// TIA Portal V17 export
// export: Created 2023-12-22T15:05:24.9190485Z, ExportSetting WithDefaults, DisplayName Totally Integrated Automation Portal, DisplayVersion V17, DisplayName TIA Portal Openness, DisplayVersion V17, DisplayName TIA Portal Version Control Interface, DisplayVersion V17, DisplayName STEP 7 Professional, DisplayVersion V17, DisplayName STEP 7 Safety, DisplayVersion V17, DisplayName WinCC Advanced, DisplayVersion V17
FUNCTION "Line_Settings" : Void   // FC2, LAD
{ S7_Optimized_Access := 'TRUE' }
VERSION : 0.1
// stored: AutoNumber true, IsIECCheckEnabled false, SetENOAutomatically false, UDAEnableTagReadback false
   VAR_INPUT
      All_lines : Int;   // Кол-во линий
   END_VAR
   VAR_IN_OUT
      Line_REQ : Int;   // Запрос линии
      Line_Now : Int;   // Линия сейчас
      Ready : Bool;   // Готовность
   END_VAR
   VAR_TEMP   // added for the SCL form of the ladder/FBD networks
      _w1 : Bool;
      _w2 : Bool;
      _w3 : Bool;
      _w4 : Bool;
      _w5 : Bool;
      _w6 : Bool;
      _w7 : Bool;
      _w8 : Bool;
      _w9 : Bool;
   END_VAR
BEGIN

REGION Network 1: Проверка корректности выбранной линии
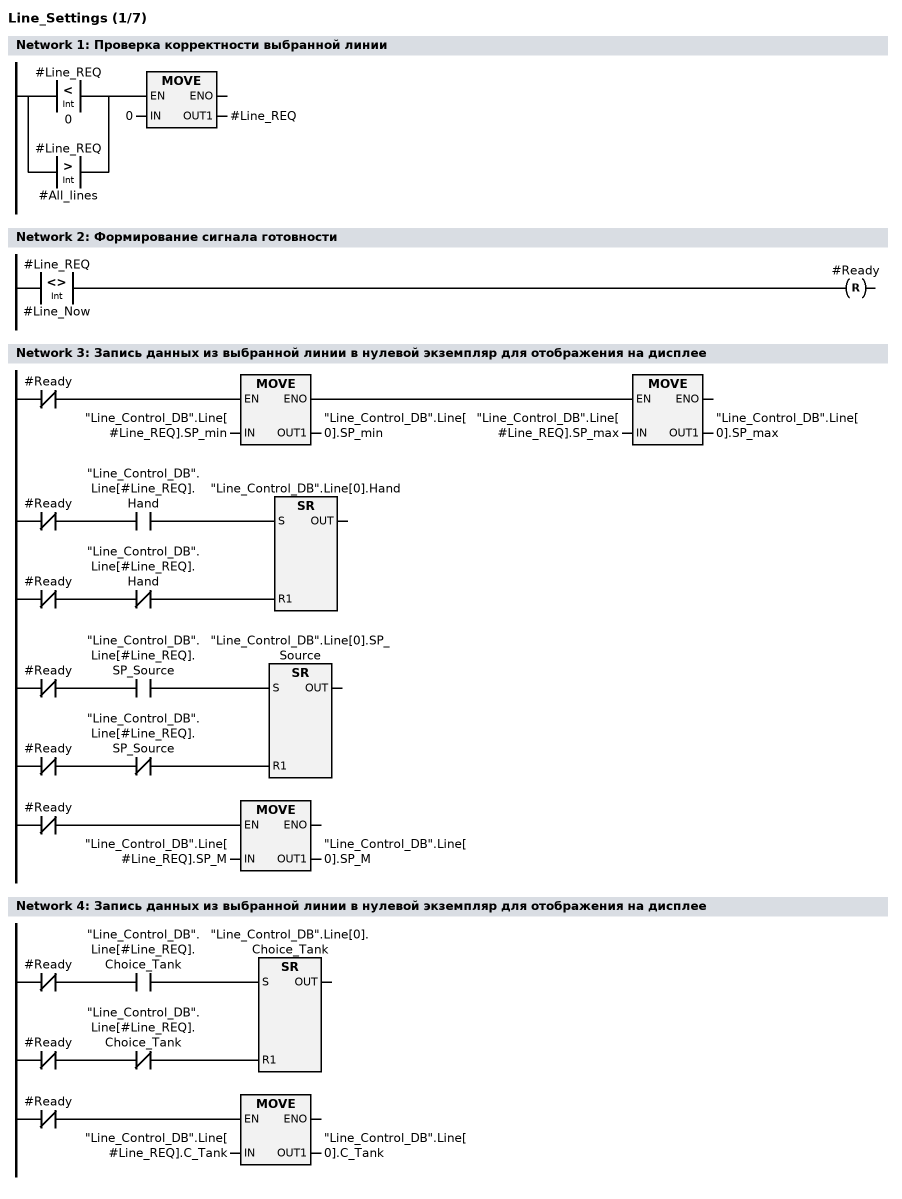
   RUNG wire#powerrail
      { S7_Templates := "SrcType := Int" } LT_Contact(in1 := #Line_REQ, in2 := 0)
      wire#w1
      Move(in := 0, out1 => #Line_REQ)
   END_RUNG
   RUNG wire#powerrail
      { S7_Templates := "SrcType := Int" } GT_Contact(in1 := #Line_REQ, in2 := #All_lines)
   END_RUNG wire#w1
   // the same network as SCL:
   IF (#Line_REQ < 0) OR (#Line_REQ > #All_lines) THEN #Line_REQ := 0; END_IF;
END_REGION

REGION Network 2: Формирование сигнала готовности
   RUNG wire#powerrail
      { S7_Templates := "SrcType := Int" } NE_Contact(in1 := #Line_REQ, in2 := #Line_Now)
      R_Coil( #Ready )
   END_RUNG
   // the same network as SCL:
   IF #Line_REQ <> #Line_Now THEN #Ready := FALSE; END_IF;
END_REGION

REGION Network 3: Запись данных из выбранной линии в нулевой экземпляр для отображения на дисплее
   RUNG wire#powerrail
      I_Contact( #Ready )
      Move(in := "Line_Control_DB".Line[#Line_REQ].SP_min, out1 => "Line_Control_DB".Line[0].SP_min)
      Move(in := "Line_Control_DB".Line[#Line_REQ].SP_max, out1 => "Line_Control_DB".Line[0].SP_max)
   END_RUNG
   RUNG wire#powerrail
      I_Contact( #Ready )
      Contact( "Line_Control_DB".Line[#Line_REQ].Hand )
      S_SR(operand := "Line_Control_DB".Line[0].Hand, r1 := wire#w1)
   END_RUNG
   RUNG wire#powerrail
      I_Contact( #Ready )
      I_Contact( "Line_Control_DB".Line[#Line_REQ].Hand )
   END_RUNG wire#w1
   RUNG wire#powerrail
      I_Contact( #Ready )
      Contact( "Line_Control_DB".Line[#Line_REQ].SP_Source )
      S_SR(operand := "Line_Control_DB".Line[0].SP_Source, r1 := wire#w2)
   END_RUNG
   RUNG wire#powerrail
      I_Contact( #Ready )
      I_Contact( "Line_Control_DB".Line[#Line_REQ].SP_Source )
   END_RUNG wire#w2
   RUNG wire#powerrail
      I_Contact( #Ready )
      Move(in := "Line_Control_DB".Line[#Line_REQ].SP_M, out1 => "Line_Control_DB".Line[0].SP_M)
   END_RUNG
   // the same network as SCL:
   IF NOT #Ready THEN
       "Line_Control_DB".Line[0].SP_min := "Line_Control_DB".Line[#Line_REQ].SP_min;
       "Line_Control_DB".Line[0].SP_max := "Line_Control_DB".Line[#Line_REQ].SP_max;
   END_IF;
   #_w1 := NOT #Ready AND NOT "Line_Control_DB".Line[#Line_REQ].Hand;
   IF NOT #Ready AND "Line_Control_DB".Line[#Line_REQ].Hand THEN
       "Line_Control_DB".Line[0].Hand := TRUE;   // SR flip-flop
   END_IF;
   IF #_w1 THEN "Line_Control_DB".Line[0].Hand := FALSE; END_IF;
   #_w2 := NOT #Ready AND NOT "Line_Control_DB".Line[#Line_REQ].SP_Source;
   IF NOT #Ready AND "Line_Control_DB".Line[#Line_REQ].SP_Source THEN
       "Line_Control_DB".Line[0].SP_Source := TRUE;   // SR flip-flop
   END_IF;
   IF #_w2 THEN "Line_Control_DB".Line[0].SP_Source := FALSE; END_IF;
   IF NOT #Ready THEN "Line_Control_DB".Line[0].SP_M := "Line_Control_DB".Line[#Line_REQ].SP_M; END_IF;
END_REGION

REGION Network 4: Запись данных из выбранной линии в нулевой экземпляр для отображения на дисплее
   RUNG wire#powerrail
      I_Contact( #Ready )
      Contact( "Line_Control_DB".Line[#Line_REQ].Choice_Tank )
      S_SR(operand := "Line_Control_DB".Line[0].Choice_Tank, r1 := wire#w1)
   END_RUNG
   RUNG wire#powerrail
      I_Contact( #Ready )
      I_Contact( "Line_Control_DB".Line[#Line_REQ].Choice_Tank )
   END_RUNG wire#w1
   RUNG wire#powerrail
      I_Contact( #Ready )
      Move(in := "Line_Control_DB".Line[#Line_REQ].C_Tank, out1 => "Line_Control_DB".Line[0].C_Tank)
   END_RUNG
   // the same network as SCL:
   #_w1 := NOT #Ready AND NOT "Line_Control_DB".Line[#Line_REQ].Choice_Tank;
   IF NOT #Ready AND "Line_Control_DB".Line[#Line_REQ].Choice_Tank THEN
       "Line_Control_DB".Line[0].Choice_Tank := TRUE;   // SR flip-flop
   END_IF;
   IF #_w1 THEN "Line_Control_DB".Line[0].Choice_Tank := FALSE; END_IF;
   IF NOT #Ready THEN "Line_Control_DB".Line[0].C_Tank := "Line_Control_DB".Line[#Line_REQ].C_Tank; END_IF;
END_REGION

REGION Network 5: Запись данных из выбранной линии в нулевой экземпляр для отображения на дисплее
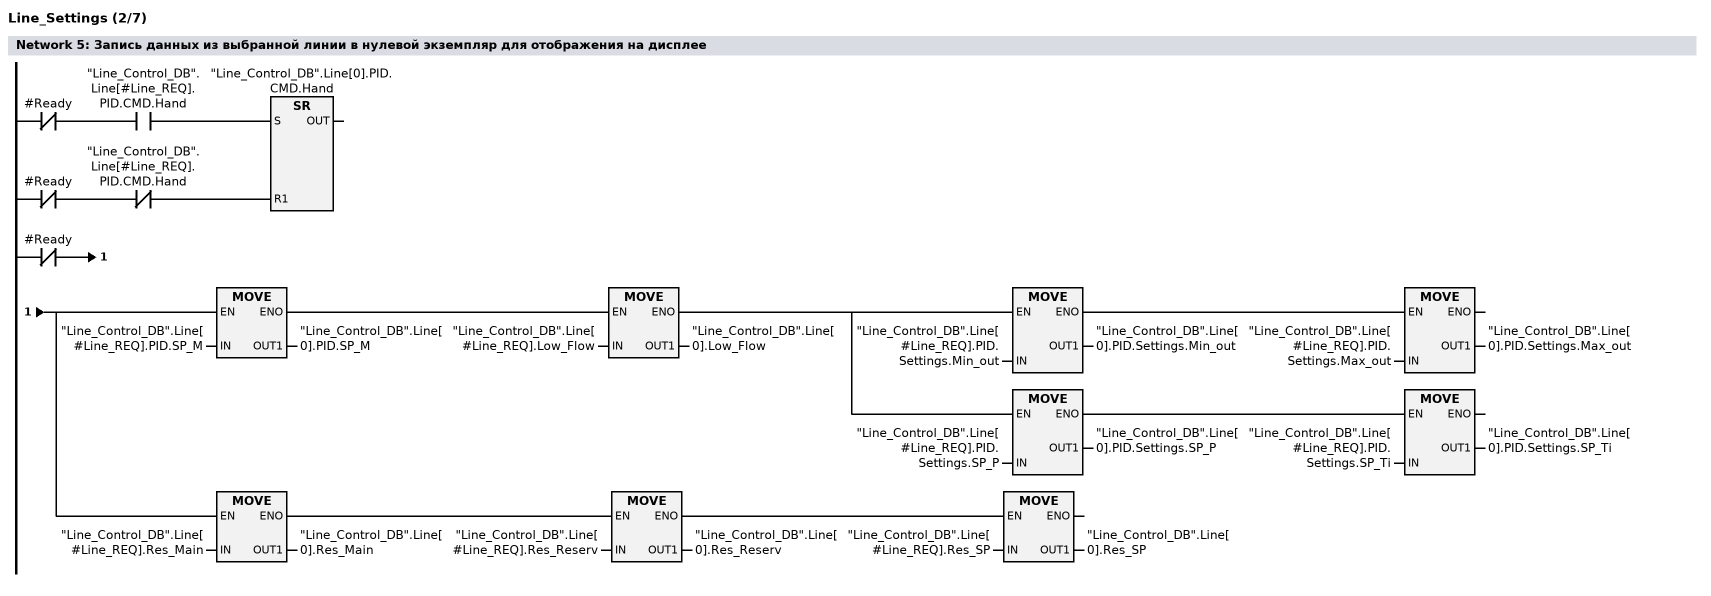
   RUNG wire#powerrail
      I_Contact( #Ready )
      Contact( "Line_Control_DB".Line[#Line_REQ].PID.CMD.Hand )
      S_SR(operand := "Line_Control_DB".Line[0].PID.CMD.Hand, r1 := wire#w1)
   END_RUNG
   RUNG wire#powerrail
      I_Contact( #Ready )
      I_Contact( "Line_Control_DB".Line[#Line_REQ].PID.CMD.Hand )
   END_RUNG wire#w1
   RUNG wire#powerrail
      I_Contact( #Ready )
      wire#w2
      Move(in := "Line_Control_DB".Line[#Line_REQ].PID.SP_M, out1 => "Line_Control_DB".Line[0].PID.SP_M)
      Move(in := "Line_Control_DB".Line[#Line_REQ].Low_Flow, out1 => "Line_Control_DB".Line[0].Low_Flow)
      wire#w3
      Move(in := "Line_Control_DB".Line[#Line_REQ].PID.Settings.Min_out, out1 => "Line_Control_DB".Line[0].PID.Settings.Min_out)
      Move(in := "Line_Control_DB".Line[#Line_REQ].PID.Settings.Max_out, out1 => "Line_Control_DB".Line[0].PID.Settings.Max_out)
   END_RUNG
   RUNG wire#w3
      Move(in := "Line_Control_DB".Line[#Line_REQ].PID.Settings.SP_P, out1 => "Line_Control_DB".Line[0].PID.Settings.SP_P)
      Move(in := "Line_Control_DB".Line[#Line_REQ].PID.Settings.SP_Ti, out1 => "Line_Control_DB".Line[0].PID.Settings.SP_Ti)
   END_RUNG
   RUNG wire#w2
      Move(in := "Line_Control_DB".Line[#Line_REQ].Res_Main, out1 => "Line_Control_DB".Line[0].Res_Main)
      Move(in := "Line_Control_DB".Line[#Line_REQ].Res_Reserv, out1 => "Line_Control_DB".Line[0].Res_Reserv)
      Move(in := "Line_Control_DB".Line[#Line_REQ].Res_SP, out1 => "Line_Control_DB".Line[0].Res_SP)
   END_RUNG
   // the same network as SCL:
   #_w1 := NOT #Ready AND NOT "Line_Control_DB".Line[#Line_REQ].PID.CMD.Hand;
   IF NOT #Ready AND "Line_Control_DB".Line[#Line_REQ].PID.CMD.Hand THEN
       "Line_Control_DB".Line[0].PID.CMD.Hand := TRUE;   // SR flip-flop
   END_IF;
   IF #_w1 THEN "Line_Control_DB".Line[0].PID.CMD.Hand := FALSE; END_IF;
   IF NOT #Ready THEN
       "Line_Control_DB".Line[0].PID.SP_M := "Line_Control_DB".Line[#Line_REQ].PID.SP_M;
       "Line_Control_DB".Line[0].Low_Flow := "Line_Control_DB".Line[#Line_REQ].Low_Flow;
       "Line_Control_DB".Line[0].PID.Settings.Min_out := "Line_Control_DB".Line[#Line_REQ].PID.Settings.Min_out;
       "Line_Control_DB".Line[0].PID.Settings.Max_out := "Line_Control_DB".Line[#Line_REQ].PID.Settings.Max_out;
       "Line_Control_DB".Line[0].PID.Settings.SP_P := "Line_Control_DB".Line[#Line_REQ].PID.Settings.SP_P;
       "Line_Control_DB".Line[0].PID.Settings.SP_Ti := "Line_Control_DB".Line[#Line_REQ].PID.Settings.SP_Ti;
       "Line_Control_DB".Line[0].Res_Main := "Line_Control_DB".Line[#Line_REQ].Res_Main;
       "Line_Control_DB".Line[0].Res_Reserv := "Line_Control_DB".Line[#Line_REQ].Res_Reserv;
       "Line_Control_DB".Line[0].Res_SP := "Line_Control_DB".Line[#Line_REQ].Res_SP;
   END_IF;
END_REGION

REGION Network 6: Запись данных из выбранной линии в нулевой экземпляр для отображения на дисплее
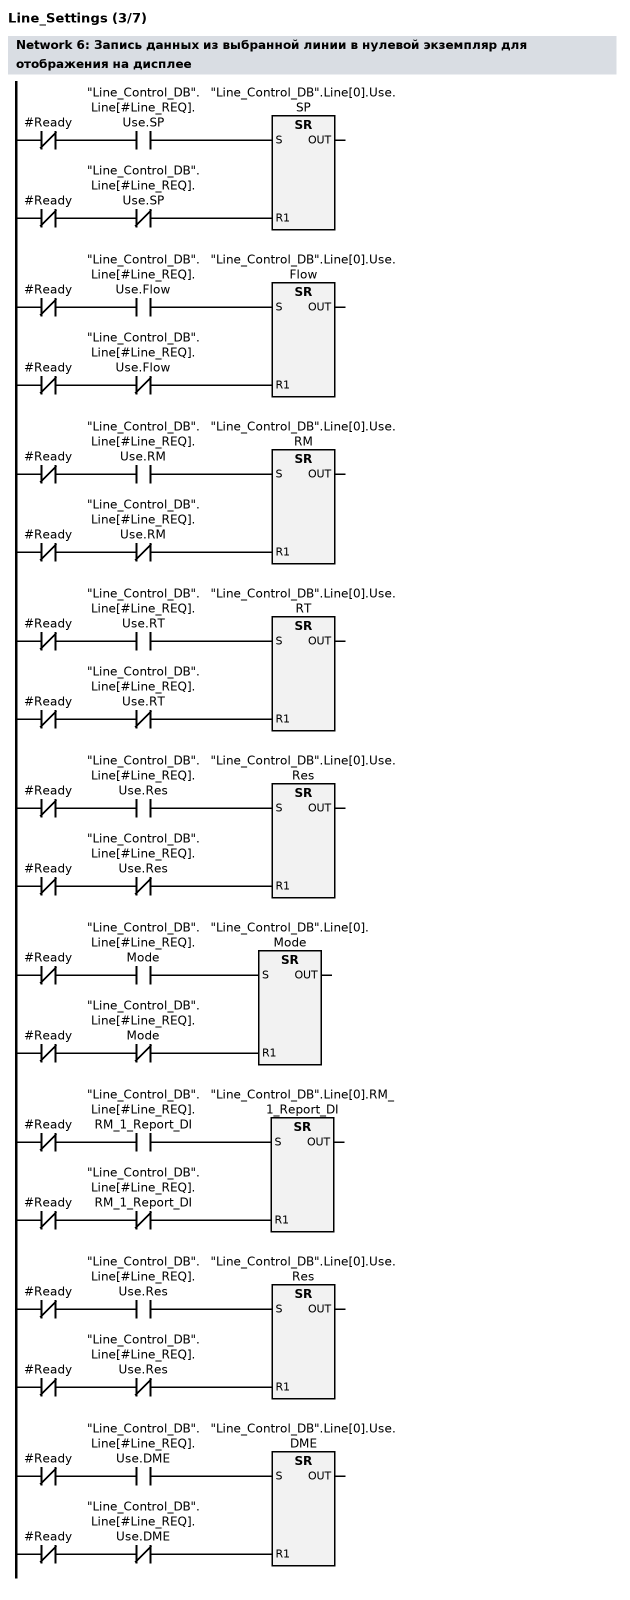
   RUNG wire#powerrail
      I_Contact( #Ready )
      Contact( "Line_Control_DB".Line[#Line_REQ].Use.SP )
      S_SR(operand := "Line_Control_DB".Line[0].Use.SP, r1 := wire#w1)
   END_RUNG
   RUNG wire#powerrail
      I_Contact( #Ready )
      I_Contact( "Line_Control_DB".Line[#Line_REQ].Use.SP )
   END_RUNG wire#w1
   RUNG wire#powerrail
      I_Contact( #Ready )
      Contact( "Line_Control_DB".Line[#Line_REQ].Use.Flow )
      S_SR(operand := "Line_Control_DB".Line[0].Use.Flow, r1 := wire#w2)
   END_RUNG
   RUNG wire#powerrail
      I_Contact( #Ready )
      I_Contact( "Line_Control_DB".Line[#Line_REQ].Use.Flow )
   END_RUNG wire#w2
   RUNG wire#powerrail
      I_Contact( #Ready )
      Contact( "Line_Control_DB".Line[#Line_REQ].Use.RM )
      S_SR(operand := "Line_Control_DB".Line[0].Use.RM, r1 := wire#w3)
   END_RUNG
   RUNG wire#powerrail
      I_Contact( #Ready )
      I_Contact( "Line_Control_DB".Line[#Line_REQ].Use.RM )
   END_RUNG wire#w3
   RUNG wire#powerrail
      I_Contact( #Ready )
      Contact( "Line_Control_DB".Line[#Line_REQ].Use.RT )
      S_SR(operand := "Line_Control_DB".Line[0].Use.RT, r1 := wire#w4)
   END_RUNG
   RUNG wire#powerrail
      I_Contact( #Ready )
      I_Contact( "Line_Control_DB".Line[#Line_REQ].Use.RT )
   END_RUNG wire#w4
   RUNG wire#powerrail
      I_Contact( #Ready )
      Contact( "Line_Control_DB".Line[#Line_REQ].Use.Res )
      S_SR(operand := "Line_Control_DB".Line[0].Use.Res, r1 := wire#w5)
   END_RUNG
   RUNG wire#powerrail
      I_Contact( #Ready )
      I_Contact( "Line_Control_DB".Line[#Line_REQ].Use.Res )
   END_RUNG wire#w5
   RUNG wire#powerrail
      I_Contact( #Ready )
      Contact( "Line_Control_DB".Line[#Line_REQ].Mode )
      S_SR(operand := "Line_Control_DB".Line[0].Mode, r1 := wire#w6)
   END_RUNG
   RUNG wire#powerrail
      I_Contact( #Ready )
      I_Contact( "Line_Control_DB".Line[#Line_REQ].Mode )
   END_RUNG wire#w6
   RUNG wire#powerrail
      I_Contact( #Ready )
      Contact( "Line_Control_DB".Line[#Line_REQ].RM_1_Report_DI )
      S_SR(operand := "Line_Control_DB".Line[0].RM_1_Report_DI, r1 := wire#w7)
   END_RUNG
   RUNG wire#powerrail
      I_Contact( #Ready )
      I_Contact( "Line_Control_DB".Line[#Line_REQ].RM_1_Report_DI )
   END_RUNG wire#w7
   RUNG wire#powerrail
      I_Contact( #Ready )
      Contact( "Line_Control_DB".Line[#Line_REQ].Use.Res )
      S_SR(operand := "Line_Control_DB".Line[0].Use.Res, r1 := wire#w8)
   END_RUNG
   RUNG wire#powerrail
      I_Contact( #Ready )
      I_Contact( "Line_Control_DB".Line[#Line_REQ].Use.Res )
   END_RUNG wire#w8
   RUNG wire#powerrail
      I_Contact( #Ready )
      Contact( "Line_Control_DB".Line[#Line_REQ].Use.DME )
      S_SR(operand := "Line_Control_DB".Line[0].Use.DME, r1 := wire#w9)
   END_RUNG
   RUNG wire#powerrail
      I_Contact( #Ready )
      I_Contact( "Line_Control_DB".Line[#Line_REQ].Use.DME )
   END_RUNG wire#w9
   // the same network as SCL:
   #_w1 := NOT #Ready AND NOT "Line_Control_DB".Line[#Line_REQ].Use.SP;
   IF NOT #Ready AND "Line_Control_DB".Line[#Line_REQ].Use.SP THEN
       "Line_Control_DB".Line[0].Use.SP := TRUE;   // SR flip-flop
   END_IF;
   IF #_w1 THEN "Line_Control_DB".Line[0].Use.SP := FALSE; END_IF;
   #_w2 := NOT #Ready AND NOT "Line_Control_DB".Line[#Line_REQ].Use.Flow;
   IF NOT #Ready AND "Line_Control_DB".Line[#Line_REQ].Use.Flow THEN
       "Line_Control_DB".Line[0].Use.Flow := TRUE;   // SR flip-flop
   END_IF;
   IF #_w2 THEN "Line_Control_DB".Line[0].Use.Flow := FALSE; END_IF;
   #_w3 := NOT #Ready AND NOT "Line_Control_DB".Line[#Line_REQ].Use.RM;
   IF NOT #Ready AND "Line_Control_DB".Line[#Line_REQ].Use.RM THEN
       "Line_Control_DB".Line[0].Use.RM := TRUE;   // SR flip-flop
   END_IF;
   IF #_w3 THEN "Line_Control_DB".Line[0].Use.RM := FALSE; END_IF;
   #_w4 := NOT #Ready AND NOT "Line_Control_DB".Line[#Line_REQ].Use.RT;
   IF NOT #Ready AND "Line_Control_DB".Line[#Line_REQ].Use.RT THEN
       "Line_Control_DB".Line[0].Use.RT := TRUE;   // SR flip-flop
   END_IF;
   IF #_w4 THEN "Line_Control_DB".Line[0].Use.RT := FALSE; END_IF;
   #_w5 := NOT #Ready AND NOT "Line_Control_DB".Line[#Line_REQ].Use.Res;
   IF NOT #Ready AND "Line_Control_DB".Line[#Line_REQ].Use.Res THEN
       "Line_Control_DB".Line[0].Use.Res := TRUE;   // SR flip-flop
   END_IF;
   IF #_w5 THEN "Line_Control_DB".Line[0].Use.Res := FALSE; END_IF;
   #_w6 := NOT #Ready AND NOT "Line_Control_DB".Line[#Line_REQ].Mode;
   IF NOT #Ready AND "Line_Control_DB".Line[#Line_REQ].Mode THEN
       "Line_Control_DB".Line[0].Mode := TRUE;   // SR flip-flop
   END_IF;
   IF #_w6 THEN "Line_Control_DB".Line[0].Mode := FALSE; END_IF;
   #_w7 := NOT #Ready AND NOT "Line_Control_DB".Line[#Line_REQ].RM_1_Report_DI;
   IF NOT #Ready AND "Line_Control_DB".Line[#Line_REQ].RM_1_Report_DI THEN
       "Line_Control_DB".Line[0].RM_1_Report_DI := TRUE;   // SR flip-flop
   END_IF;
   IF #_w7 THEN "Line_Control_DB".Line[0].RM_1_Report_DI := FALSE; END_IF;
   #_w8 := NOT #Ready AND NOT "Line_Control_DB".Line[#Line_REQ].Use.Res;
   IF NOT #Ready AND "Line_Control_DB".Line[#Line_REQ].Use.Res THEN
       "Line_Control_DB".Line[0].Use.Res := TRUE;   // SR flip-flop
   END_IF;
   IF #_w8 THEN "Line_Control_DB".Line[0].Use.Res := FALSE; END_IF;
   #_w9 := NOT #Ready AND NOT "Line_Control_DB".Line[#Line_REQ].Use.DME;
   IF NOT #Ready AND "Line_Control_DB".Line[#Line_REQ].Use.DME THEN
       "Line_Control_DB".Line[0].Use.DME := TRUE;   // SR flip-flop
   END_IF;
   IF #_w9 THEN "Line_Control_DB".Line[0].Use.DME := FALSE; END_IF;
END_REGION

REGION Network 7: Запись данных из выбранной линии в нулевой экземпляр для отображения на дисплее
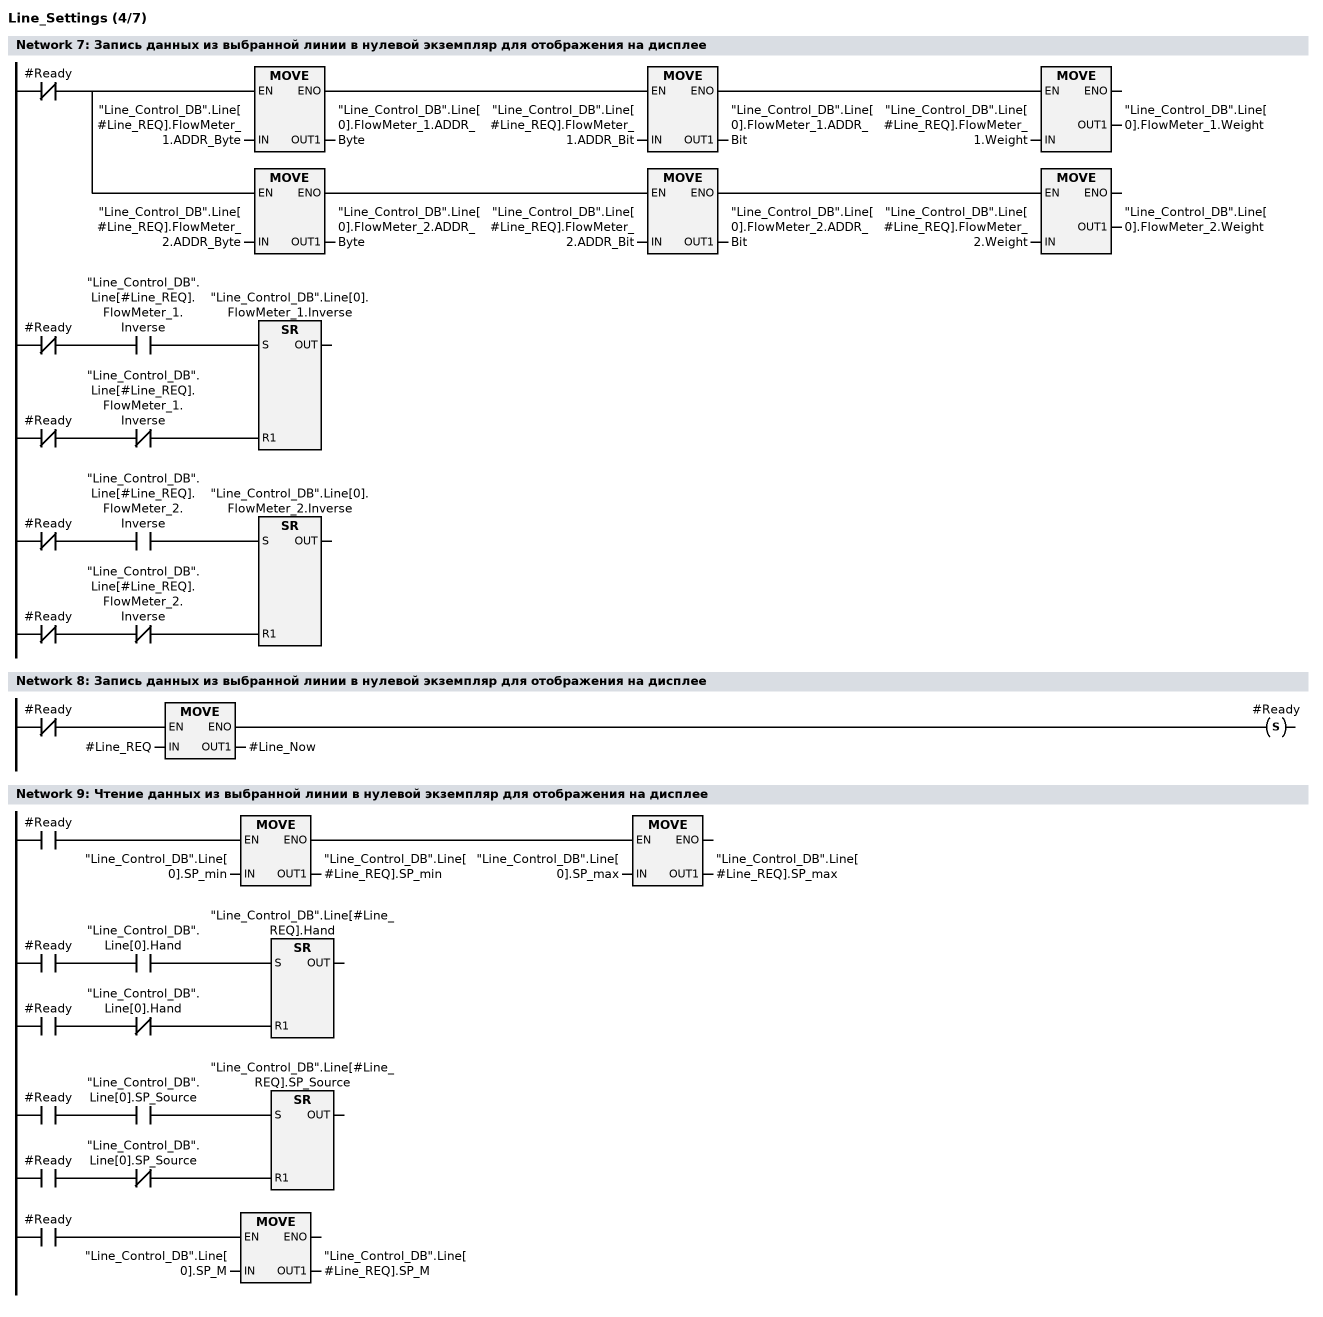
   RUNG wire#powerrail
      I_Contact( #Ready )
      wire#w1
      Move(in := "Line_Control_DB".Line[#Line_REQ].FlowMeter_1.ADDR_Byte, out1 => "Line_Control_DB".Line[0].FlowMeter_1.ADDR_Byte)
      Move(in := "Line_Control_DB".Line[#Line_REQ].FlowMeter_1.ADDR_Bit, out1 => "Line_Control_DB".Line[0].FlowMeter_1.ADDR_Bit)
      Move(in := "Line_Control_DB".Line[#Line_REQ].FlowMeter_1.Weight, out1 => "Line_Control_DB".Line[0].FlowMeter_1.Weight)
   END_RUNG
   RUNG wire#w1
      Move(in := "Line_Control_DB".Line[#Line_REQ].FlowMeter_2.ADDR_Byte, out1 => "Line_Control_DB".Line[0].FlowMeter_2.ADDR_Byte)
      Move(in := "Line_Control_DB".Line[#Line_REQ].FlowMeter_2.ADDR_Bit, out1 => "Line_Control_DB".Line[0].FlowMeter_2.ADDR_Bit)
      Move(in := "Line_Control_DB".Line[#Line_REQ].FlowMeter_2.Weight, out1 => "Line_Control_DB".Line[0].FlowMeter_2.Weight)
   END_RUNG
   RUNG wire#powerrail
      I_Contact( #Ready )
      Contact( "Line_Control_DB".Line[#Line_REQ].FlowMeter_1.Inverse )
      S_SR(operand := "Line_Control_DB".Line[0].FlowMeter_1.Inverse, r1 := wire#w2)
   END_RUNG
   RUNG wire#powerrail
      I_Contact( #Ready )
      I_Contact( "Line_Control_DB".Line[#Line_REQ].FlowMeter_1.Inverse )
   END_RUNG wire#w2
   RUNG wire#powerrail
      I_Contact( #Ready )
      Contact( "Line_Control_DB".Line[#Line_REQ].FlowMeter_2.Inverse )
      S_SR(operand := "Line_Control_DB".Line[0].FlowMeter_2.Inverse, r1 := wire#w3)
   END_RUNG
   RUNG wire#powerrail
      I_Contact( #Ready )
      I_Contact( "Line_Control_DB".Line[#Line_REQ].FlowMeter_2.Inverse )
   END_RUNG wire#w3
   // the same network as SCL:
   IF NOT #Ready THEN
       "Line_Control_DB".Line[0].FlowMeter_1.ADDR_Byte := "Line_Control_DB".Line[#Line_REQ].FlowMeter_1.ADDR_Byte;
       "Line_Control_DB".Line[0].FlowMeter_1.ADDR_Bit := "Line_Control_DB".Line[#Line_REQ].FlowMeter_1.ADDR_Bit;
       "Line_Control_DB".Line[0].FlowMeter_1.Weight := "Line_Control_DB".Line[#Line_REQ].FlowMeter_1.Weight;
       "Line_Control_DB".Line[0].FlowMeter_2.ADDR_Byte := "Line_Control_DB".Line[#Line_REQ].FlowMeter_2.ADDR_Byte;
       "Line_Control_DB".Line[0].FlowMeter_2.ADDR_Bit := "Line_Control_DB".Line[#Line_REQ].FlowMeter_2.ADDR_Bit;
       "Line_Control_DB".Line[0].FlowMeter_2.Weight := "Line_Control_DB".Line[#Line_REQ].FlowMeter_2.Weight;
   END_IF;
   #_w1 := NOT #Ready AND NOT "Line_Control_DB".Line[#Line_REQ].FlowMeter_1.Inverse;
   IF NOT #Ready AND "Line_Control_DB".Line[#Line_REQ].FlowMeter_1.Inverse THEN
       "Line_Control_DB".Line[0].FlowMeter_1.Inverse := TRUE;   // SR flip-flop
   END_IF;
   IF #_w1 THEN "Line_Control_DB".Line[0].FlowMeter_1.Inverse := FALSE; END_IF;
   #_w2 := NOT #Ready AND NOT "Line_Control_DB".Line[#Line_REQ].FlowMeter_2.Inverse;
   IF NOT #Ready AND "Line_Control_DB".Line[#Line_REQ].FlowMeter_2.Inverse THEN
       "Line_Control_DB".Line[0].FlowMeter_2.Inverse := TRUE;   // SR flip-flop
   END_IF;
   IF #_w2 THEN "Line_Control_DB".Line[0].FlowMeter_2.Inverse := FALSE; END_IF;
END_REGION

REGION Network 8: Запись данных из выбранной линии в нулевой экземпляр для отображения на дисплее
   RUNG wire#powerrail
      I_Contact( #Ready )
      Move(in := #Line_REQ, out1 => #Line_Now)
      S_Coil( #Ready )
   END_RUNG
   // the same network as SCL:
   IF NOT #Ready THEN
       #Line_Now := #Line_REQ;
       #Ready := TRUE;
   END_IF;
END_REGION

REGION Network 9: Чтение данных из выбранной линии в нулевой экземпляр для отображения на дисплее
   RUNG wire#powerrail
      Contact( #Ready )
      Move(in := "Line_Control_DB".Line[0].SP_min, out1 => "Line_Control_DB".Line[#Line_REQ].SP_min)
      Move(in := "Line_Control_DB".Line[0].SP_max, out1 => "Line_Control_DB".Line[#Line_REQ].SP_max)
   END_RUNG
   RUNG wire#powerrail
      Contact( #Ready )
      Contact( "Line_Control_DB".Line[0].Hand )
      S_SR(operand := "Line_Control_DB".Line[#Line_REQ].Hand, r1 := wire#w1)
   END_RUNG
   RUNG wire#powerrail
      Contact( #Ready )
      I_Contact( "Line_Control_DB".Line[0].Hand )
   END_RUNG wire#w1
   RUNG wire#powerrail
      Contact( #Ready )
      Contact( "Line_Control_DB".Line[0].SP_Source )
      S_SR(operand := "Line_Control_DB".Line[#Line_REQ].SP_Source, r1 := wire#w2)
   END_RUNG
   RUNG wire#powerrail
      Contact( #Ready )
      I_Contact( "Line_Control_DB".Line[0].SP_Source )
   END_RUNG wire#w2
   RUNG wire#powerrail
      Contact( #Ready )
      Move(in := "Line_Control_DB".Line[0].SP_M, out1 => "Line_Control_DB".Line[#Line_REQ].SP_M)
   END_RUNG
   // the same network as SCL:
   IF #Ready THEN
       "Line_Control_DB".Line[#Line_REQ].SP_min := "Line_Control_DB".Line[0].SP_min;
       "Line_Control_DB".Line[#Line_REQ].SP_max := "Line_Control_DB".Line[0].SP_max;
   END_IF;
   #_w1 := #Ready AND NOT "Line_Control_DB".Line[0].Hand;
   IF #Ready AND "Line_Control_DB".Line[0].Hand THEN
       "Line_Control_DB".Line[#Line_REQ].Hand := TRUE;   // SR flip-flop
   END_IF;
   IF #_w1 THEN "Line_Control_DB".Line[#Line_REQ].Hand := FALSE; END_IF;
   #_w2 := #Ready AND NOT "Line_Control_DB".Line[0].SP_Source;
   IF #Ready AND "Line_Control_DB".Line[0].SP_Source THEN
       "Line_Control_DB".Line[#Line_REQ].SP_Source := TRUE;   // SR flip-flop
   END_IF;
   IF #_w2 THEN "Line_Control_DB".Line[#Line_REQ].SP_Source := FALSE; END_IF;
   IF #Ready THEN "Line_Control_DB".Line[#Line_REQ].SP_M := "Line_Control_DB".Line[0].SP_M; END_IF;
END_REGION

REGION Network 10: Чтение данных из выбранной линии в нулевой экземпляр для отображения на дисплее
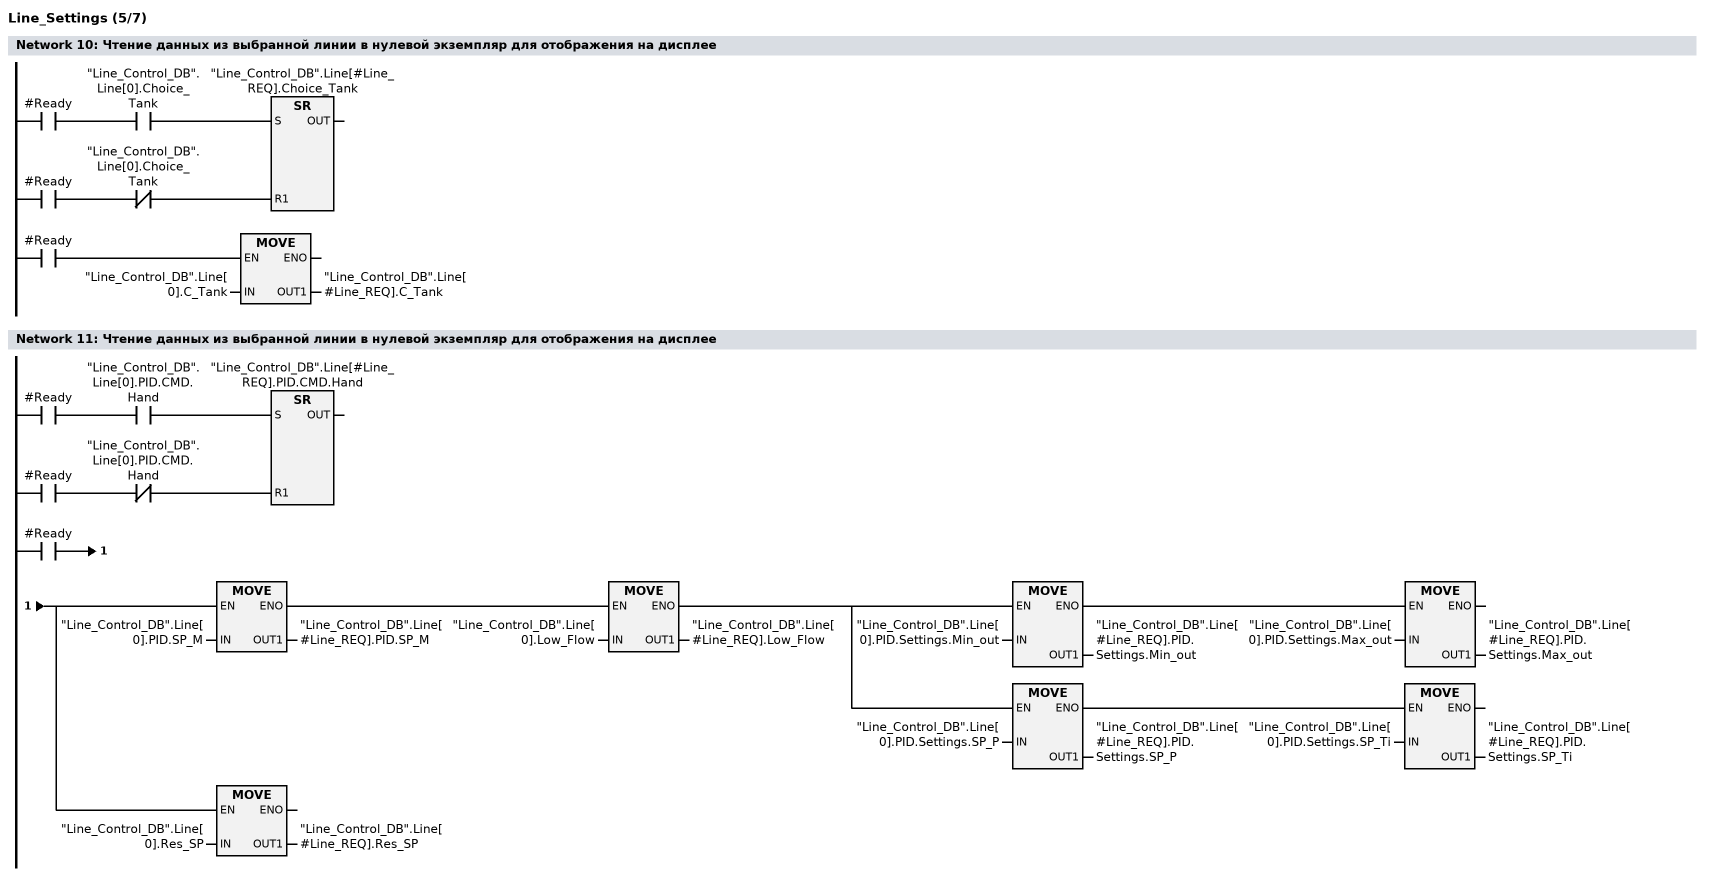
   RUNG wire#powerrail
      Contact( #Ready )
      Contact( "Line_Control_DB".Line[0].Choice_Tank )
      S_SR(operand := "Line_Control_DB".Line[#Line_REQ].Choice_Tank, r1 := wire#w1)
   END_RUNG
   RUNG wire#powerrail
      Contact( #Ready )
      I_Contact( "Line_Control_DB".Line[0].Choice_Tank )
   END_RUNG wire#w1
   RUNG wire#powerrail
      Contact( #Ready )
      Move(in := "Line_Control_DB".Line[0].C_Tank, out1 => "Line_Control_DB".Line[#Line_REQ].C_Tank)
   END_RUNG
   // the same network as SCL:
   #_w1 := #Ready AND NOT "Line_Control_DB".Line[0].Choice_Tank;
   IF #Ready AND "Line_Control_DB".Line[0].Choice_Tank THEN
       "Line_Control_DB".Line[#Line_REQ].Choice_Tank := TRUE;   // SR flip-flop
   END_IF;
   IF #_w1 THEN "Line_Control_DB".Line[#Line_REQ].Choice_Tank := FALSE; END_IF;
   IF #Ready THEN "Line_Control_DB".Line[#Line_REQ].C_Tank := "Line_Control_DB".Line[0].C_Tank; END_IF;
END_REGION

REGION Network 11: Чтение данных из выбранной линии в нулевой экземпляр для отображения на дисплее
   RUNG wire#powerrail
      Contact( #Ready )
      Contact( "Line_Control_DB".Line[0].PID.CMD.Hand )
      S_SR(operand := "Line_Control_DB".Line[#Line_REQ].PID.CMD.Hand, r1 := wire#w1)
   END_RUNG
   RUNG wire#powerrail
      Contact( #Ready )
      I_Contact( "Line_Control_DB".Line[0].PID.CMD.Hand )
   END_RUNG wire#w1
   RUNG wire#powerrail
      Contact( #Ready )
      wire#w2
      Move(in := "Line_Control_DB".Line[0].PID.SP_M, out1 => "Line_Control_DB".Line[#Line_REQ].PID.SP_M)
      Move(in := "Line_Control_DB".Line[0].Low_Flow, out1 => "Line_Control_DB".Line[#Line_REQ].Low_Flow)
      wire#w3
      Move(in := "Line_Control_DB".Line[0].PID.Settings.Min_out, out1 => "Line_Control_DB".Line[#Line_REQ].PID.Settings.Min_out)
      Move(in := "Line_Control_DB".Line[0].PID.Settings.Max_out, out1 => "Line_Control_DB".Line[#Line_REQ].PID.Settings.Max_out)
   END_RUNG
   RUNG wire#w3
      Move(in := "Line_Control_DB".Line[0].PID.Settings.SP_P, out1 => "Line_Control_DB".Line[#Line_REQ].PID.Settings.SP_P)
      Move(in := "Line_Control_DB".Line[0].PID.Settings.SP_Ti, out1 => "Line_Control_DB".Line[#Line_REQ].PID.Settings.SP_Ti)
   END_RUNG
   RUNG wire#w2
      Move(in := "Line_Control_DB".Line[0].Res_SP, out1 => "Line_Control_DB".Line[#Line_REQ].Res_SP)
   END_RUNG
   // the same network as SCL:
   #_w1 := #Ready AND NOT "Line_Control_DB".Line[0].PID.CMD.Hand;
   IF #Ready AND "Line_Control_DB".Line[0].PID.CMD.Hand THEN
       "Line_Control_DB".Line[#Line_REQ].PID.CMD.Hand := TRUE;   // SR flip-flop
   END_IF;
   IF #_w1 THEN "Line_Control_DB".Line[#Line_REQ].PID.CMD.Hand := FALSE; END_IF;
   IF #Ready THEN
       "Line_Control_DB".Line[#Line_REQ].PID.SP_M := "Line_Control_DB".Line[0].PID.SP_M;
       "Line_Control_DB".Line[#Line_REQ].Low_Flow := "Line_Control_DB".Line[0].Low_Flow;
       "Line_Control_DB".Line[#Line_REQ].PID.Settings.Min_out := "Line_Control_DB".Line[0].PID.Settings.Min_out;
       "Line_Control_DB".Line[#Line_REQ].PID.Settings.Max_out := "Line_Control_DB".Line[0].PID.Settings.Max_out;
       "Line_Control_DB".Line[#Line_REQ].PID.Settings.SP_P := "Line_Control_DB".Line[0].PID.Settings.SP_P;
       "Line_Control_DB".Line[#Line_REQ].PID.Settings.SP_Ti := "Line_Control_DB".Line[0].PID.Settings.SP_Ti;
       "Line_Control_DB".Line[#Line_REQ].Res_SP := "Line_Control_DB".Line[0].Res_SP;
   END_IF;
END_REGION

REGION Network 12: Чтение данных из выбранной линии в нулевой экземпляр для отображения на дисплее
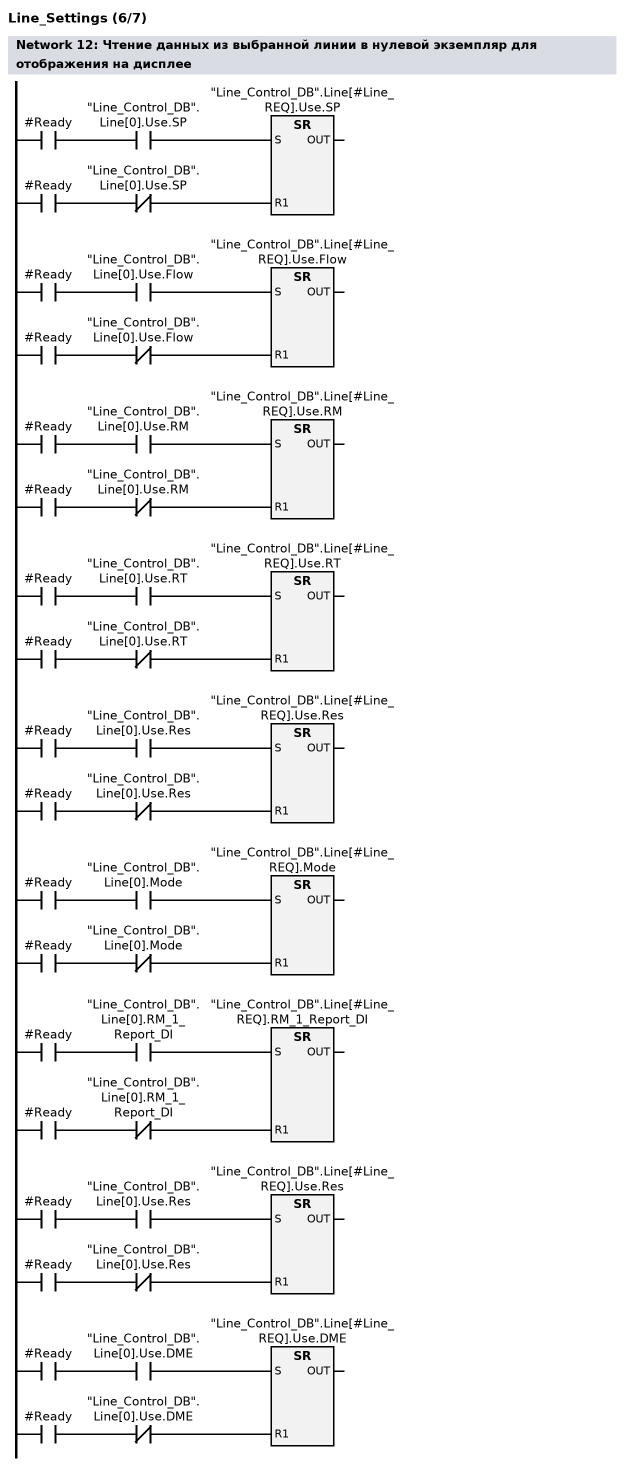
   RUNG wire#powerrail
      Contact( #Ready )
      Contact( "Line_Control_DB".Line[0].Use.SP )
      S_SR(operand := "Line_Control_DB".Line[#Line_REQ].Use.SP, r1 := wire#w1)
   END_RUNG
   RUNG wire#powerrail
      Contact( #Ready )
      I_Contact( "Line_Control_DB".Line[0].Use.SP )
   END_RUNG wire#w1
   RUNG wire#powerrail
      Contact( #Ready )
      Contact( "Line_Control_DB".Line[0].Use.Flow )
      S_SR(operand := "Line_Control_DB".Line[#Line_REQ].Use.Flow, r1 := wire#w2)
   END_RUNG
   RUNG wire#powerrail
      Contact( #Ready )
      I_Contact( "Line_Control_DB".Line[0].Use.Flow )
   END_RUNG wire#w2
   RUNG wire#powerrail
      Contact( #Ready )
      Contact( "Line_Control_DB".Line[0].Use.RM )
      S_SR(operand := "Line_Control_DB".Line[#Line_REQ].Use.RM, r1 := wire#w3)
   END_RUNG
   RUNG wire#powerrail
      Contact( #Ready )
      I_Contact( "Line_Control_DB".Line[0].Use.RM )
   END_RUNG wire#w3
   RUNG wire#powerrail
      Contact( #Ready )
      Contact( "Line_Control_DB".Line[0].Use.RT )
      S_SR(operand := "Line_Control_DB".Line[#Line_REQ].Use.RT, r1 := wire#w4)
   END_RUNG
   RUNG wire#powerrail
      Contact( #Ready )
      I_Contact( "Line_Control_DB".Line[0].Use.RT )
   END_RUNG wire#w4
   RUNG wire#powerrail
      Contact( #Ready )
      Contact( "Line_Control_DB".Line[0].Use.Res )
      S_SR(operand := "Line_Control_DB".Line[#Line_REQ].Use.Res, r1 := wire#w5)
   END_RUNG
   RUNG wire#powerrail
      Contact( #Ready )
      I_Contact( "Line_Control_DB".Line[0].Use.Res )
   END_RUNG wire#w5
   RUNG wire#powerrail
      Contact( #Ready )
      Contact( "Line_Control_DB".Line[0].Mode )
      S_SR(operand := "Line_Control_DB".Line[#Line_REQ].Mode, r1 := wire#w6)
   END_RUNG
   RUNG wire#powerrail
      Contact( #Ready )
      I_Contact( "Line_Control_DB".Line[0].Mode )
   END_RUNG wire#w6
   RUNG wire#powerrail
      Contact( #Ready )
      Contact( "Line_Control_DB".Line[0].RM_1_Report_DI )
      S_SR(operand := "Line_Control_DB".Line[#Line_REQ].RM_1_Report_DI, r1 := wire#w7)
   END_RUNG
   RUNG wire#powerrail
      Contact( #Ready )
      I_Contact( "Line_Control_DB".Line[0].RM_1_Report_DI )
   END_RUNG wire#w7
   RUNG wire#powerrail
      Contact( #Ready )
      Contact( "Line_Control_DB".Line[0].Use.Res )
      S_SR(operand := "Line_Control_DB".Line[#Line_REQ].Use.Res, r1 := wire#w8)
   END_RUNG
   RUNG wire#powerrail
      Contact( #Ready )
      I_Contact( "Line_Control_DB".Line[0].Use.Res )
   END_RUNG wire#w8
   RUNG wire#powerrail
      Contact( #Ready )
      Contact( "Line_Control_DB".Line[0].Use.DME )
      S_SR(operand := "Line_Control_DB".Line[#Line_REQ].Use.DME, r1 := wire#w9)
   END_RUNG
   RUNG wire#powerrail
      Contact( #Ready )
      I_Contact( "Line_Control_DB".Line[0].Use.DME )
   END_RUNG wire#w9
   // the same network as SCL:
   #_w1 := #Ready AND NOT "Line_Control_DB".Line[0].Use.SP;
   IF #Ready AND "Line_Control_DB".Line[0].Use.SP THEN
       "Line_Control_DB".Line[#Line_REQ].Use.SP := TRUE;   // SR flip-flop
   END_IF;
   IF #_w1 THEN "Line_Control_DB".Line[#Line_REQ].Use.SP := FALSE; END_IF;
   #_w2 := #Ready AND NOT "Line_Control_DB".Line[0].Use.Flow;
   IF #Ready AND "Line_Control_DB".Line[0].Use.Flow THEN
       "Line_Control_DB".Line[#Line_REQ].Use.Flow := TRUE;   // SR flip-flop
   END_IF;
   IF #_w2 THEN "Line_Control_DB".Line[#Line_REQ].Use.Flow := FALSE; END_IF;
   #_w3 := #Ready AND NOT "Line_Control_DB".Line[0].Use.RM;
   IF #Ready AND "Line_Control_DB".Line[0].Use.RM THEN
       "Line_Control_DB".Line[#Line_REQ].Use.RM := TRUE;   // SR flip-flop
   END_IF;
   IF #_w3 THEN "Line_Control_DB".Line[#Line_REQ].Use.RM := FALSE; END_IF;
   #_w4 := #Ready AND NOT "Line_Control_DB".Line[0].Use.RT;
   IF #Ready AND "Line_Control_DB".Line[0].Use.RT THEN
       "Line_Control_DB".Line[#Line_REQ].Use.RT := TRUE;   // SR flip-flop
   END_IF;
   IF #_w4 THEN "Line_Control_DB".Line[#Line_REQ].Use.RT := FALSE; END_IF;
   #_w5 := #Ready AND NOT "Line_Control_DB".Line[0].Use.Res;
   IF #Ready AND "Line_Control_DB".Line[0].Use.Res THEN
       "Line_Control_DB".Line[#Line_REQ].Use.Res := TRUE;   // SR flip-flop
   END_IF;
   IF #_w5 THEN "Line_Control_DB".Line[#Line_REQ].Use.Res := FALSE; END_IF;
   #_w6 := #Ready AND NOT "Line_Control_DB".Line[0].Mode;
   IF #Ready AND "Line_Control_DB".Line[0].Mode THEN
       "Line_Control_DB".Line[#Line_REQ].Mode := TRUE;   // SR flip-flop
   END_IF;
   IF #_w6 THEN "Line_Control_DB".Line[#Line_REQ].Mode := FALSE; END_IF;
   #_w7 := #Ready AND NOT "Line_Control_DB".Line[0].RM_1_Report_DI;
   IF #Ready AND "Line_Control_DB".Line[0].RM_1_Report_DI THEN
       "Line_Control_DB".Line[#Line_REQ].RM_1_Report_DI := TRUE;   // SR flip-flop
   END_IF;
   IF #_w7 THEN "Line_Control_DB".Line[#Line_REQ].RM_1_Report_DI := FALSE; END_IF;
   #_w8 := #Ready AND NOT "Line_Control_DB".Line[0].Use.Res;
   IF #Ready AND "Line_Control_DB".Line[0].Use.Res THEN
       "Line_Control_DB".Line[#Line_REQ].Use.Res := TRUE;   // SR flip-flop
   END_IF;
   IF #_w8 THEN "Line_Control_DB".Line[#Line_REQ].Use.Res := FALSE; END_IF;
   #_w9 := #Ready AND NOT "Line_Control_DB".Line[0].Use.DME;
   IF #Ready AND "Line_Control_DB".Line[0].Use.DME THEN
       "Line_Control_DB".Line[#Line_REQ].Use.DME := TRUE;   // SR flip-flop
   END_IF;
   IF #_w9 THEN "Line_Control_DB".Line[#Line_REQ].Use.DME := FALSE; END_IF;
END_REGION

REGION Network 13: Чтение данных из выбранной линии в нулевой экземпляр для отображения на дисплее
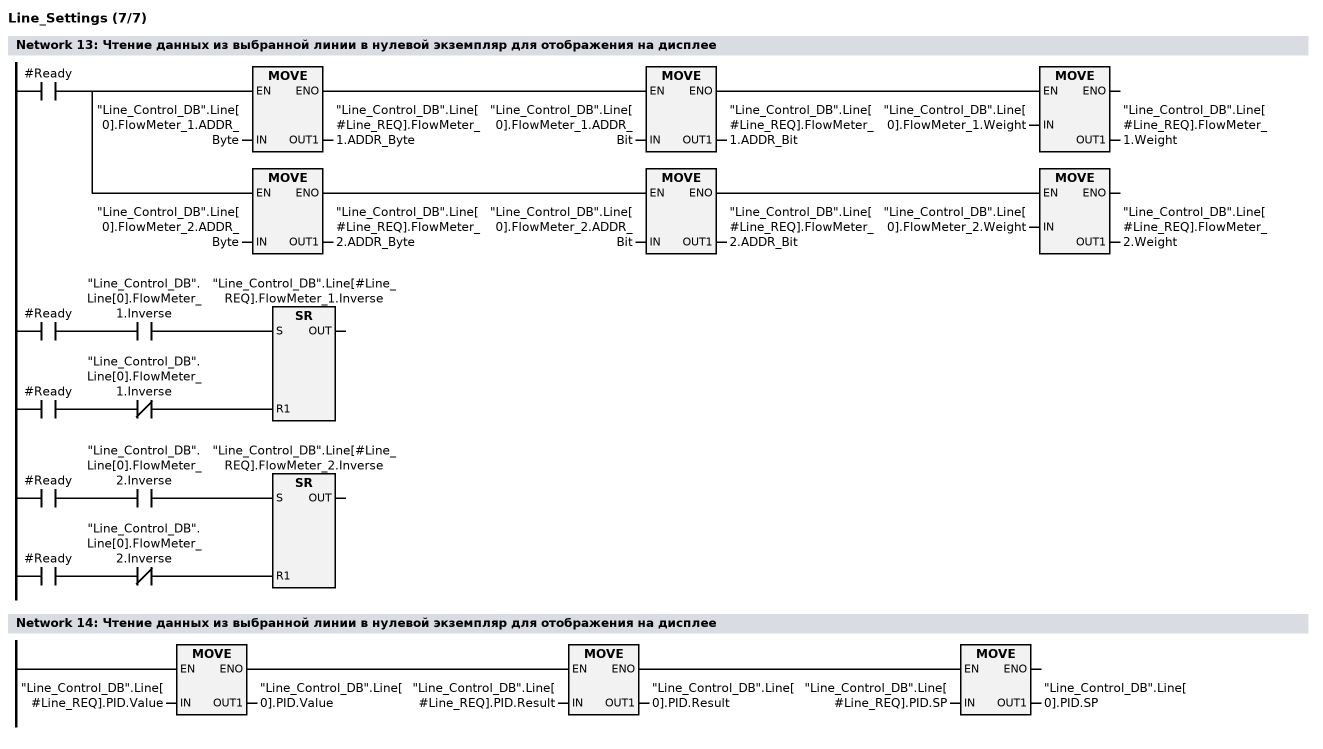
   RUNG wire#powerrail
      Contact( #Ready )
      wire#w1
      Move(in := "Line_Control_DB".Line[0].FlowMeter_1.ADDR_Byte, out1 => "Line_Control_DB".Line[#Line_REQ].FlowMeter_1.ADDR_Byte)
      Move(in := "Line_Control_DB".Line[0].FlowMeter_1.ADDR_Bit, out1 => "Line_Control_DB".Line[#Line_REQ].FlowMeter_1.ADDR_Bit)
      Move(in := "Line_Control_DB".Line[0].FlowMeter_1.Weight, out1 => "Line_Control_DB".Line[#Line_REQ].FlowMeter_1.Weight)
   END_RUNG
   RUNG wire#w1
      Move(in := "Line_Control_DB".Line[0].FlowMeter_2.ADDR_Byte, out1 => "Line_Control_DB".Line[#Line_REQ].FlowMeter_2.ADDR_Byte)
      Move(in := "Line_Control_DB".Line[0].FlowMeter_2.ADDR_Bit, out1 => "Line_Control_DB".Line[#Line_REQ].FlowMeter_2.ADDR_Bit)
      Move(in := "Line_Control_DB".Line[0].FlowMeter_2.Weight, out1 => "Line_Control_DB".Line[#Line_REQ].FlowMeter_2.Weight)
   END_RUNG
   RUNG wire#powerrail
      Contact( #Ready )
      Contact( "Line_Control_DB".Line[0].FlowMeter_1.Inverse )
      S_SR(operand := "Line_Control_DB".Line[#Line_REQ].FlowMeter_1.Inverse, r1 := wire#w2)
   END_RUNG
   RUNG wire#powerrail
      Contact( #Ready )
      I_Contact( "Line_Control_DB".Line[0].FlowMeter_1.Inverse )
   END_RUNG wire#w2
   RUNG wire#powerrail
      Contact( #Ready )
      Contact( "Line_Control_DB".Line[0].FlowMeter_2.Inverse )
      S_SR(operand := "Line_Control_DB".Line[#Line_REQ].FlowMeter_2.Inverse, r1 := wire#w3)
   END_RUNG
   RUNG wire#powerrail
      Contact( #Ready )
      I_Contact( "Line_Control_DB".Line[0].FlowMeter_2.Inverse )
   END_RUNG wire#w3
   // the same network as SCL:
   IF #Ready THEN
       "Line_Control_DB".Line[#Line_REQ].FlowMeter_1.ADDR_Byte := "Line_Control_DB".Line[0].FlowMeter_1.ADDR_Byte;
       "Line_Control_DB".Line[#Line_REQ].FlowMeter_1.ADDR_Bit := "Line_Control_DB".Line[0].FlowMeter_1.ADDR_Bit;
       "Line_Control_DB".Line[#Line_REQ].FlowMeter_1.Weight := "Line_Control_DB".Line[0].FlowMeter_1.Weight;
       "Line_Control_DB".Line[#Line_REQ].FlowMeter_2.ADDR_Byte := "Line_Control_DB".Line[0].FlowMeter_2.ADDR_Byte;
       "Line_Control_DB".Line[#Line_REQ].FlowMeter_2.ADDR_Bit := "Line_Control_DB".Line[0].FlowMeter_2.ADDR_Bit;
       "Line_Control_DB".Line[#Line_REQ].FlowMeter_2.Weight := "Line_Control_DB".Line[0].FlowMeter_2.Weight;
   END_IF;
   #_w1 := #Ready AND NOT "Line_Control_DB".Line[0].FlowMeter_1.Inverse;
   IF #Ready AND "Line_Control_DB".Line[0].FlowMeter_1.Inverse THEN
       "Line_Control_DB".Line[#Line_REQ].FlowMeter_1.Inverse := TRUE;   // SR flip-flop
   END_IF;
   IF #_w1 THEN "Line_Control_DB".Line[#Line_REQ].FlowMeter_1.Inverse := FALSE; END_IF;
   #_w2 := #Ready AND NOT "Line_Control_DB".Line[0].FlowMeter_2.Inverse;
   IF #Ready AND "Line_Control_DB".Line[0].FlowMeter_2.Inverse THEN
       "Line_Control_DB".Line[#Line_REQ].FlowMeter_2.Inverse := TRUE;   // SR flip-flop
   END_IF;
   IF #_w2 THEN "Line_Control_DB".Line[#Line_REQ].FlowMeter_2.Inverse := FALSE; END_IF;
END_REGION

REGION Network 14: Чтение данных из выбранной линии в нулевой экземпляр для отображения на дисплее
   RUNG wire#powerrail
      Move(in := "Line_Control_DB".Line[#Line_REQ].PID.Value, out1 => "Line_Control_DB".Line[0].PID.Value)
      Move(in := "Line_Control_DB".Line[#Line_REQ].PID.Result, out1 => "Line_Control_DB".Line[0].PID.Result)
      Move(in := "Line_Control_DB".Line[#Line_REQ].PID.SP, out1 => "Line_Control_DB".Line[0].PID.SP)
   END_RUNG
   // the same network as SCL:
   "Line_Control_DB".Line[0].PID.Value := "Line_Control_DB".Line[#Line_REQ].PID.Value;
   "Line_Control_DB".Line[0].PID.Result := "Line_Control_DB".Line[#Line_REQ].PID.Result;
   "Line_Control_DB".Line[0].PID.SP := "Line_Control_DB".Line[#Line_REQ].PID.SP;
END_REGION
END_FUNCTION
